{region '#Template'}
	{attribute 'Version' := '1.2.2.0'}
	{attribute 'Tags' := '"LCID": "1031", "Text": "General, Cabinet, Control cabinet, Event groups, Categories, Notification classes, Event classes"'}
	{attribute 'Tags' := '"LCID": "1033", "Text": "General, Cabinet, Control cabinet, Event groups, Categories, Notification classes, Event classes"'}
	{attribute 'Using' := '"Type": "Template", "URI": "EC_AMEV"'}
	{attribute 'Description' := '"LCID": "1031", "Text": "Ereignisgruppen, Kategorien"'}
	{attribute 'Description' := '"LCID": "1033", "Text": "Event groups, categories"'}
{endregion}
FUNCTION_BLOCK FB_BA_EvtGroups EXTENDS FB_BA_View
VAR_INPUT CONSTANT
	LifeSafety						: FB_BA_EvtCategory;
	SafetyMsg						: FB_BA_EvtCategory;
	AlarmMsg						: FB_BA_EvtCategory;
	FaultMsg						: FB_BA_EvtCategory;
	MaintenanceMsg01				: FB_BA_EvtCategory;
	MaintenanceMsg02				: FB_BA_EvtCategory;
	SystemMsg						: FB_BA_EvtCategory;
	ManualOp						: FB_BA_EvtCategory;
	OtherMsg						: FB_BA_EvtCategory;
END_VAR

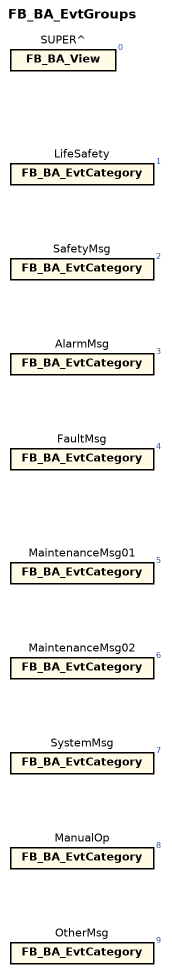
SUPER^(); // FB_BA_View
LifeSafety(); // FB_BA_EvtCategory
SafetyMsg(); // FB_BA_EvtCategory
AlarmMsg(); // FB_BA_EvtCategory
FaultMsg(); // FB_BA_EvtCategory
MaintenanceMsg01(); // FB_BA_EvtCategory
MaintenanceMsg02(); // FB_BA_EvtCategory
SystemMsg(); // FB_BA_EvtCategory
ManualOp(); // FB_BA_EvtCategory
OtherMsg(); // FB_BA_EvtCategory

METHOD FB_init : BOOL
VAR_INPUT
	bInitRetains : BOOL; // if TRUE, the retain variables are initialized (warm start / cold start)
	bInCopyCode : BOOL;  // if TRUE, the instance afterwards gets moved into the copy code (online change)
END_VAR
//===================================================================
// Ereigniskategorie - Gefahr für Leben // Event category - Danger to life
// Brandalarm, Überfall // Fire alarm, robbery
LifeSafety.iParent							:= THIS^;
LifeSafety.iLabel							:= LblControl_EvtCategoryLifeSafty;									  
LifeSafety.sObjectName						:= '{Idx=01}';
LifeSafety.eDPADMode						:= E_BA_DPADMode.eInclude;																						
LifeSafety.EC.nInstanceID						:= EC_ID.NC10;
LifeSafety.EC.sObjectName						:= '{Idx=10}';
LifeSafety.EC.eEventType						:= E_BA_EventType.eAlarm;
LifeSafety.EC.aPriority[1]						:= 10;
LifeSafety.EC.aPriority[2]						:= 11;
LifeSafety.EC.aPriority[3]						:= 12;
LifeSafety.EC.eAlarmMode						:= E_BA_AlarmMode.eExtended;	//Erweiterter Alarm
//===================================================================		
// Ereigniskategorie - Gefahrenmeldung, Sicherheitsmeldung // Event category - hazard alert, safety message
// Einbruch, unberechtigter Zutritt // Burglary, unauthorised entry
SafetyMsg.iParent							:= THIS^;
SafetyMsg.iLabel							:= LblControl_EvtCategorySaftyMessage;									  
SafetyMsg.sObjectName						:= '{Idx=01}';
SafetyMsg.eDPADMode							:= E_BA_DPADMode.eInclude;																						
SafetyMsg.EC.nInstanceID						:= EC_ID.NC20;
SafetyMsg.EC.sObjectName						:= '{Idx=20}';
SafetyMsg.EC.eEventType							:= E_BA_EventType.eAlarm;
SafetyMsg.EC.aPriority[1]						:= 40;
SafetyMsg.EC.aPriority[2]						:= 41;
SafetyMsg.EC.aPriority[3]						:= 42;
SafetyMsg.EC.eAlarmMode						:= E_BA_AlarmMode.eExtended;	//Erweiterter Alarm

//===================================================================//
// Ereigniskategorie - Alarmeldung - Meldung signalisiert Anlagenausfall oder erfordert sofortigen Eingriff 
// Event category - Alarm message - Message signals system failure or requires immediate intervention 
// Sicherheitstemperaturbegrenzer (STB), Sicherheitsdruckbegrenzer (SDB), Übertemperatur der Warmwasserbereitung (WWB), Sicherheitsventile, Hauptpumpen, Keilriemenwächter, Frequenzumformer, Kälteanlagen, Spannungsausfall usw
// Safety temperature limiter, safety pressure limiter, excess temperature of water heating, safety valves, main pumps, V-belt monitors, frequency converters, refrigeration systems, voltage failure, etc.
AlarmMsg.iParent							:= THIS^;
AlarmMsg.iLabel								:= LblControl_EvtCategoryAlarmMessage;									  
AlarmMsg.sObjectName						:= '{Idx=01}';
AlarmMsg.eDPADMode							:= E_BA_DPADMode.eInclude;																						
AlarmMsg.EC.nInstanceID							:= EC_ID.NC30;
AlarmMsg.EC.sObjectName							:= '{Idx=30}';
AlarmMsg.EC.eEventType							:= E_BA_EventType.eAlarm;
AlarmMsg.EC.aPriority[1]						:= 70;
AlarmMsg.EC.aPriority[2]						:= 71;
AlarmMsg.EC.aPriority[3]						:= 72;
AlarmMsg.EC.eAlarmMode						:= E_BA_AlarmMode.eExtended;	//Erweiterter Alarm


//===================================================================
// Ereigniskategorie - Störungsmeldung - Meldung weist auf einen anormalen Betriebszustand hin
// Event category - malfunction message - message indicates abnormal operating condition
// Temperaturwächter (TW), Druckwächter (DW), Temperaturüberwachung von Wärmetauscher (WT) und WWB, Motorschutz, Aufzug-Sammelstörmeldung, Netzdrücke usw.
// Temperature monitor, pressure monitor, temperature monitoring of heat exchanger and water heating, motor protection, lift collective fault signal, mains pressures, etc.
FaultMsg.iParent							:= THIS^;
FaultMsg.iLabel								:= LblControl_EvtCategoryFaultMessage;							  
FaultMsg.sObjectName						:= '{Idx=01}';
FaultMsg.eDPADMode							:= E_BA_DPADMode.eInclude;																						
FaultMsg.EC.nInstanceID							:= EC_ID.NC40;
FaultMsg.EC.sObjectName							:= '{Idx=40}';
FaultMsg.EC.eEventType							:= E_BA_EventType.eDisturb;
FaultMsg.EC.aPriority[1]						:= 100;
FaultMsg.EC.aPriority[2]						:= 101;
FaultMsg.EC.aPriority[3]						:= 102;
FaultMsg.EC.eAlarmMode						:= E_BA_AlarmMode.eStandard;	//Standard Alarm
//===================================================================
// Ereigniskategorie - Wartungsmeldung, Hinweis auf Wartungsaktivität o.ä.
// Event category - Maintenance message Maintenance message, indication of maintenance activity or similar.
// Betriebsstunden, Behälterstand, Reparaturschalter usw.
// Operating hours, tank level, repair switch, etc.
MaintenanceMsg01.iParent					:= THIS^;
MaintenanceMsg01.iLabel						:= LblControl_EvtCategoryMaintenanceMessage;									  
MaintenanceMsg01.sObjectName				:= '{Idx=01}';
MaintenanceMsg01.eDPADMode					:= E_BA_DPADMode.eInclude;																						
MaintenanceMsg01.EC.nInstanceID					:= EC_ID.NC50;
MaintenanceMsg01.EC.sObjectName					:= '{Idx=50}';
MaintenanceMsg01.EC.eEventType					:= E_BA_EventType.eMaintenance;
MaintenanceMsg01.EC.aPriority[1]				:= 130;
MaintenanceMsg01.EC.aPriority[2]				:= 131;
MaintenanceMsg01.EC.aPriority[3]				:= 132;
MaintenanceMsg01.EC.eAlarmMode						:= E_BA_AlarmMode.eStandard;	//Standard Alarm

// Filterende erreicht, Filter verschmutzt usw.
// Filter end reached, filter dirty, etc.
MaintenanceMsg02.iParent					:= THIS^;
MaintenanceMsg02.iLabel						:= LblControl_EvtCategoryMaintenanceMessage;									  
MaintenanceMsg02.sObjectName				:= '{Idx=02}';
MaintenanceMsg02.sDescription				:= '{Wartungsmeldung}';
MaintenanceMsg02.eDPADMode					:= E_BA_DPADMode.eInclude;																						
MaintenanceMsg02.EC.nInstanceID					:= EC_ID.NC51;
MaintenanceMsg02.EC.sObjectName					:= '{Idx=51}';
MaintenanceMsg02.EC.eEventType					:= E_BA_EventType.eAlarm;
MaintenanceMsg02.EC.aPriority[1]				:= 135;
MaintenanceMsg02.EC.aPriority[2]				:= 136;
MaintenanceMsg02.EC.aPriority[3]				:= 137;
MaintenanceMsg02.EC.eAlarmMode						:= E_BA_AlarmMode.eStandard;	//Standard Alarm
//===================================================================
//===================================================================
// Ereigniskategorie - Systemmeldung, Störungsmeldung aus GA-System
// Event category - System message, System message, Fault message from building automation system
// Gerätestörung, Batteriemeldung, Kommunikationsunterbrechung usw.
// Unit malfunction, battery message, communication interruption, etc.
SystemMsg.iParent							:= THIS^;
SystemMsg.iLabel							:= LblControl_EvtCategorySystem;									  
SystemMsg.sObjectName						:= '{Idx=01}';
SystemMsg.eDPADMode							:= E_BA_DPADMode.eInclude;																						
SystemMsg.EC.nInstanceID						:= EC_ID.NC60;
SystemMsg.EC.sObjectName						:= '{Idx=60}';
SystemMsg.EC.eEventType							:= E_BA_EventType.eNotification;
SystemMsg.EC.aPriority[1]						:= 180;
SystemMsg.EC.aPriority[2]						:= 181;
SystemMsg.EC.aPriority[3]						:= 182;
SystemMsg.EC.eAlarmMode						:= E_BA_AlarmMode.eSimple;	//Simple Alarm
//===================================================================//
//	Ereigniskategorie - Manual operation, Handeingriff
ManualOp.iParent							:= THIS^;
ManualOp.iLabel						 		:= LblControl_EvtCategoryManualOperation;									  
ManualOp.sObjectName						:= '{Idx=01}';
ManualOp.eDPADMode							:= E_BA_DPADMode.eInclude;																						
ManualOp.EC.nInstanceID							:= EC_ID.NC70;
ManualOp.EC.sObjectName							:= '{Idx=70}';
ManualOp.EC.eEventType							:= E_BA_EventType.eAlarm;
ManualOp.EC.aPriority[1]						:= 220;
ManualOp.EC.aPriority[2]						:= 220;
ManualOp.EC.aPriority[3]						:= 220;
ManualOp.EC.eAlarmMode						:= E_BA_AlarmMode.eSimple;	//Simple Alarm
//===================================================================//
// Ereigniskategorie - Freibleibend, Sonstige Meldungen
// Event category - Other message, Not binding, Other messages
// Betriebszustandswechsel, Betriebsarten, Trendspeicher voll usw.
// Operating status change, operating modes, trend memory full, etc.
OtherMsg.iParent							:= THIS^;
OtherMsg.iLabel						 		:= LblControl_EvtCategoryOther;									  
OtherMsg.sObjectName						:= '{Idx=01}';
OtherMsg.eDPADMode							:= E_BA_DPADMode.eInclude;																						
OtherMsg.EC.nInstanceID							:= EC_ID.NC80;
OtherMsg.EC.sObjectName							:= '{Idx=80}';
OtherMsg.EC.eEventType							:= E_BA_EventType.eAlarm;
OtherMsg.EC.aPriority[1]						:= 230;
OtherMsg.EC.aPriority[2]						:= 231;
OtherMsg.EC.aPriority[3]						:= 232;
OtherMsg.EC.eAlarmMode						:= E_BA_AlarmMode.eSimple;	//Simple Alarm
END_METHOD

END_FUNCTION_BLOCK

(* stored: Version 1.1.0.1, ProductVersion 3.1.4024.9
   POU FB_BA_EvtGroups: Id {a16d9c8f-b06b-4288-928b-c49f378d4c72}, SpecialFunc None
   Method FB_init: Id {141e99f7-1b1d-4ee4-ad95-1ce93fecd9b1} *)
